Omron CX-Programmer project NewProject (CX-Programmer 9.61)

# PLC SILO_SIMULATION: CP1E N20

## Global symbols (name address type ; comment)
0.00 BOOL  ; B START
0.01 BOOL  ; B STOP
0.04 BOOL  ; MODE A
0.05 BOOL  ; MODE B
0.07 BOOL  ; TOR
100.02 BOOL  ; L RUN
200.00 BOOL  ; I R

## Program NewProgram1 (cyclic task 0)

### Section Section1

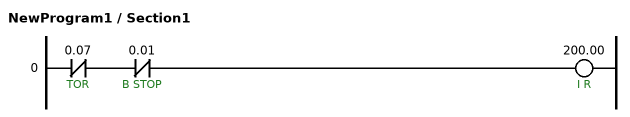
; rung 0
LDNOT 0.07  ; TOR
ANDNOT 0.01  ; B STOP
OUT 200.00  ; I R

### Section END
; rung 0
END(001)